PROGRAM prgInflux
VAR
	_influx : fbInfluxPerformanceLogging;
END_VAR

_influx();

END_PROGRAM

(* stored: Version 1.1.0.1, ProductVersion 3.1.4024.3
   POU prgInflux: Id {17e948a9-7828-4cea-9f14-e278446d659c}, SpecialFunc None *)
